VISUALIZATION Pendant  // 1024x768
END_VISUALIZATION

(* stored: Version 1.1.0.1, ProductVersion 3.1.4024.15
   Visu Pendant: Id {ccc5429d-fd15-4b7a-9efe-a44c0e8de7e0} *)
